TYPE (* DataPanel Modules with medium IO density DI Struct *)
  (* Version 1.0, 2025-07-21, franz *)
  PACKAGE DataPanel::io::MI::DI;
  DataPanel_MI_DI_S : STRUCT
    Pin : USINT := 255;
  END_STRUCT;
END_TYPE
